INTERFACE I_AnalogScale EXTENDS I_TransformLrealValue

PROPERTY InputMaximum : LREAL
GET
END_GET
SET
END_SET
END_PROPERTY

PROPERTY InputMinimum : LREAL
GET
END_GET
SET
END_SET
END_PROPERTY

PROPERTY OutputMaximum : LREAL
GET
END_GET
SET
END_SET
END_PROPERTY

PROPERTY OutputMinimum : LREAL
GET
END_GET
SET
END_SET
END_PROPERTY

END_INTERFACE

(* stored: Version 1.1.0.1, ProductVersion 3.1.4026.18
   Itf I_AnalogScale: Id {e3f6f230-57c3-4b01-86fd-9afa774b2c71}
   Property InputMaximum: Id {e9792567-ace9-4c7c-9ea3-de7ee35eded7}
   Get Get: Id {10d77b64-987d-47b3-882a-1f371629d2c7}
   Set Set: Id {9e3f0a21-b7b3-4e24-8217-08d2c73282aa}
   Property InputMinimum: Id {9cb5a823-8101-4614-a784-4d966af483ef}
   Get Get: Id {9c9270fd-c1ff-4ef5-8ff5-3ec9a82cfa68}
   Set Set: Id {cd786c49-edc2-4e2e-922f-6f5a516fac42}
   Property OutputMaximum: Id {b142b85a-91be-4563-a07c-51f713596441}
   Get Get: Id {12c1dfbc-f316-4a2f-b0aa-aa75ef8b8fa9}
   Set Set: Id {97de8491-496c-4e14-a8a9-58f98202ab6e}
   Property OutputMinimum: Id {52547ed7-964e-4526-97b4-0ae37e9f8a41}
   Get Get: Id {e90ebef2-5a8d-4a13-9070-0a23a1a98121}
   Set Set: Id {cf1adeab-61b6-4bf4-9b27-df00c7039758} *)
